(* PLC project  *)

CONFIGURATION Empty_Module_15
END_CONFIGURATION
